Yaskawa INFORM job: R1_W53-A4(90,0)R2.JBI

/JOB
//NAME R1_W53-A4(90,0)R2
///FOLDERNAME KRIS-SCIANA
//POS
///NPOS 18,18,0,0,0,0
///TOOL 0
///POSTYPE PULSE
///PULSE
C00000=120458,47711,-19664,-12728,104208,-22558
C00001=128682,99899,51858,-38063,102058,-11895
C00002=125592,100494,53893,-37558,100021,-12435
C00003=117769,53841,-3568,-7004,89352,-33862
C00004=118319,55966,-2495,-7211,89822,-33727
C00005=127393,85542,37674,-37833,96354,-10529
C00006=118983,88052,33036,-15664,100505,-10201
C00007=114637,82539,25445,-1803,99860,-9026
C00008=114316,82458,25346,-216,99794,-11375
C00009=114685,80246,17709,-453,103292,-11364
C00010=115098,70838,11827,1692,99842,-11617
C00011=113736,75911,18067,1996,98640,-12045
C00012=113399,77247,19724,2086,98314,-12154
C00013=113713,72298,10773,2034,101271,-12011
C00014=113713,72392,10731,2035,101345,-12010
C00015=113713,82237,8364,2107,107857,-11898
C00016=113713,94041,8886,2043,74694,-11800
C00017=69402,82237,8364,2107,68954,-11898
BC00000=269740,485755,1075175
BC00001=264781,512151,1075175
BC00002=264781,512151,1075175
BC00003=264644,511631,1075175
BC00004=264644,511631,1075175
BC00005=264781,512151,1075175
BC00006=264781,512151,1075175
BC00007=264781,512151,1075175
BC00008=264781,512151,1075175
BC00009=264781,512151,1075175
BC00010=264782,512151,1075173
BC00011=264782,512150,1075171
BC00012=264782,512151,1075173
BC00013=264782,512151,1075173
BC00014=264782,512151,1075173
BC00015=264782,512151,1075173
BC00016=242210,512151,1075173
BC00017=139527,574913,1075173
//INST
///DATE 2023/12/05 10:28
///ATTR SC,RW
///GROUP1 RB1,BS1
NOP
'Path S1026
SFTOF
MOVL C00000 BC00000 V=1000.0
MOVL C00001 BC00001 V=83.3
MOVL C00002 BC00002 V=50.0
REFP 1 C00003 BC00003
REFP 2 C00004 BC00004
MACRO1 MJ#(0) ARGF7
ARCON
MOVL C00005 BC00005 V=8.3
MOVL C00006 BC00006 V=8.3
MOVL C00007 BC00007 V=8.3
MOVL C00008 BC00008 V=8.3
ARCOF
MOVL C00009 BC00009 V=83.3
MOVL C00010 BC00010 V=83.3
ARCON
MOVL C00011 BC00011 V=8.3
MOVL C00012 BC00012 V=8.3
ARCOF
MOVL C00013 BC00013 V=83.3
MOVJ C00014 BC00014 VJ=50.00
MOVJ C00015 BC00015 VJ=50.00
MOVJ C00016 BC00016 VJ=50.00
MOVJ C00017 BC00017 VJ=50.00
SFTOF
'
END
